INTERFACE I_SimpleLogMessage EXTENDS I_Base

{attribute 'monitoring':='call'}
PROPERTY Message : T_MaxString
GET
END_GET
END_PROPERTY

{attribute 'monitoring':='call'}
PROPERTY Severity : USINT
GET
END_GET
END_PROPERTY

END_INTERFACE

(* stored: Version 1.1.0.1
   Itf I_SimpleLogMessage: Id {b12f37b1-a322-467e-a88e-610ceb5c6fd8}
   Property Message: Id {15e99c4c-d6ce-499a-830c-259ea98a550e}
   Get Get: Id {9844eb0b-ec54-41bb-9b6e-3446d0e0b6d3}
   Property Severity: Id {9025d844-05e8-4a77-a081-00eef6b4dd86}
   Get Get: Id {2aafae57-15c3-4f90-a4fc-f03330fc8181} *)
